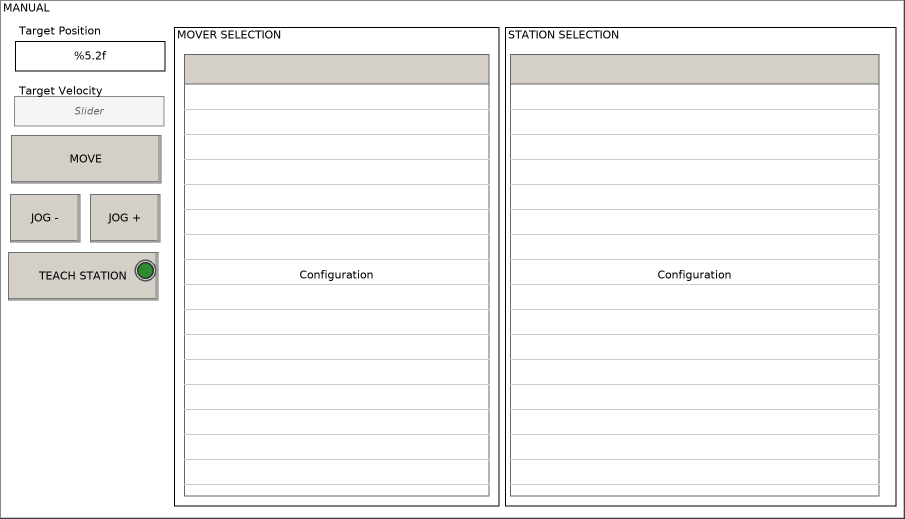
VISUALIZATION VI_XTSManualVisu  // 905x519
VAR_IN_OUT
	xts : XTS_System;
END_VAR
VAR
	stTableStruct : ARRAY [1..25] OF stTableStructx10;
END_VAR
    Rectangle (0,0 905x519), "MANUAL"
    Button (11,135 150x48), "MOVE"
        tap xts.bManualMove
    Button (10,194 70x48), "JOG -"
        tap xts.bJogBackwards
    Button (90,194 70x48), "JOG +"
        tap xts.bJogForward
    Slider (14,96 150x30), variable: xts.lrTargetVelocity, scale 1..4000
    Label (16,76 150x30), "Target Velocity"
    Rectangle (15,41 150x30), "%5.2f", text variable: xts.lrTargetPosition, input disabled if: xts.udiStationSelection<>0
        OnMouseClick: write the text variable via Default
    Label (16,16 150x30), "Target Position"
    Button (8,252 150x48), "TEACH STATION", input disabled if: xts.iVisuMoverSelection<1
        tap xts.bTeachStation
    Lamp1 (133,256 25x29), variable: xts.bTeachDone, style: Lamp-Lamp1-Green
    Rectangle (174,27 325x479), "MOVER SELECTION"
    Table (184,54 305x442), "Configuration", data array: stTableStruct
        p1137915858: xts.iVisuMoverSelection
        p3854506369: xts.ax[INDEX].ax.NcToPlc.AxisId
        p1892666644: xts.ax[INDEX].ax.NcToPlc.ModuloSetPos
        p338671338: xts.ax[INDEX].ax.NcToPlc.SetVelo
        p2170511999: xts.ax[INDEX].ax.Status.MotionState
        p3723444502: xts.ax[INDEX].ax.NcToPlc.ErrorCode
        p2232123230: Name
        p511219082: Position
        p1755163831: Velocity
        p2237128397: Error ID
        p505689113: Process Time
        p1757482276: Stop Positions
        p4088588272: Ack Mode
        p2243050616: Disable
        p516019884: Travel Time
        p2685023577: stTableStruct.b1
        p3312258591: stTableStruct.b2
        p1791247317: stTableStruct.b3
        p262371475: stTableStruct.b4
        p4008173056: stTableStruct.b5
        p2340480326: stTableStruct.b6
        p606709900: stTableStruct.b7
        p1095668682: stTableStruct.b8
        p1037165547: stTableStruct.b9
        p1488378029: stTableStruct.b10
        Columns.Column.[3].Template: OnMouseClick: write the text variable via Default
        Columns.Column.[8].Template: xts.aStations[INDEX].stCfg.bDisable=true; toggle xts.aStations[INDEX].stCfg.bDisable
        Columns.Column.[6].Template: OnMouseClick: write the text variable via Default, min 1, max 3
        Columns.Column.[4].Template: OnMouseClick: write the text variable via Default
        Columns.Column.[5].Template: OnMouseClick: write the text variable via Default
        Columns.Column.[0].Template: OnMouseClick: OpenDialog Dialog=Mover_VISU, Parameters={fbMover: xts.aMovers[INDEX]}, OpenModal=True, OpenCentered=True
        Columns.Column.[7].Template: OnMouseClick: write the text variable via Default
        Columns.Column.[9].Template: OnMouseClick: write the text variable via Default
    Rectangle (505,27 391x479), "STATION SELECTION"
    Table (510,54 369x442), "Configuration", data array: stTableStruct
        p3854506369: xts.stCfg.stStationsCfg[INDEX].sName
        p1892666644: xts.stCfg.stStationsCfg[INDEX].lrStartPosition
        p338671338: xts.stCfg.stStationsCfg[INDEX].lrStopPosition[1]
        p2170511999: xts.stCfg.stStationsCfg[INDEX].lrStopPosition[2]
        p3723444502: xts.stCfg.stStationsCfg[INDEX].lrStopPosition[3]
        p1218418051: xts.stCfg.stStationsCfg[INDEX].lrProcessingTime
        p746581629: xts.stCfg.stStationsCfg[INDEX].uiNumStopPositions
        p3104783080: xts.stCfg.stStationsCfg[INDEX].lrTravelTime
        p7306298: xts.stCfg.stStationsCfg[INDEX].lrEndPosition
        p511219082: Start Position
        p1755163831: Stop Position 1
        p4092479075: Stop Position 2
        p2237128397: Stop Position 3
        p505689113: Process Time
        p1757482276: Stop Positions
        p4088588272: Travel Time
        p2243050616: Extra Cfg.
        p516019884: End Position
        p2685023577: stTableStruct.b1
        p3312258591: stTableStruct.b2
        p1791247317: stTableStruct.b3
        p262371475: stTableStruct.b4
        p4008173056: stTableStruct.b5
        p2340480326: stTableStruct.b6
        p606709900: stTableStruct.b7
        p1095668682: stTableStruct.b8
        p1037165547: stTableStruct.b9
        p1488378029: stTableStruct.b10
        p1137915858: xts.iVisuStationSelection
        p1420305297: xts.iVisuStopPositionSelection
        Columns.Column.[6].Template: OnMouseClick: write the text variable via Default, min 1, max 3
        Columns.Column.[5].Template: OnMouseClick: write the text variable via Default
        Columns.Column.[7].Template: OnMouseClick: write the text variable via Default
        Columns.Column.[9].Template: OnMouseClick: write the text variable via Default
        Columns.Column.[1].Template: OnMouseClick: write the text variable via Default
END_VISUALIZATION

(* stored: Version 1.1.0.1, ProductVersion 3.1.4024.11
   Visu VI_XTSManualVisu: Id {8e157e60-4eff-4fe8-ae62-1eabfb57ca5c} *)
